INTERFACE I_PackML_AbortingCommands

METHOD StateComplete
VAR_INPUT
END_VAR
END_METHOD

END_INTERFACE

(* stored: Version 1.1.0.1, ProductVersion 3.1.4024.12
   Itf I_PackML_AbortingCommands: Id {d9a12bf1-10a0-0e97-0748-591bd5c252aa}
   Method StateComplete: Id {3ca7c5f9-823e-0bc5-2d60-2d304ba6d2d0} *)
